(* IEC 61131-3 sources: AXOpen/src/components.festo.drives/ctrl/src/AxoCmmtAs (part 2) *)

                    IF Parametrization.Outputs.Done AND NOT Parametrization.Outputs.Error THEN
                        State := UINT#48;
                    END_IF;
                    IF Parametrization.Outputs.Error THEN
                        Messenger.Activate( UINT#1456, eAxoMessageCategory#Error);
                        MC_HomeErrorID :=   DINT#1456;
                        State := UINT#59;
                    END_IF;
                END_IF;
                IF State = UINT#48 THEN
                    Busy := TRUE;
                    Active := TRUE;
                    Parametrization.Inputs.Enable := FALSE;
                    IF  NOT Parametrization.Outputs.Done THEN
                        State := UINT#49;
                    END_IF;
                END_IF;
                //Write  PNU 11735 Homing mode
                IF State = UINT#49 THEN
                    Busy := TRUE;
                    Active := TRUE;
                    Parametrization.Inputs.Enable := TRUE;
                    Parametrization.Inputs.ReadWrite   := TRUE;
                    Parametrization.Inputs.ParameterNo := 11735;//mode
                    Parametrization.Inputs.Subindex    := 0;
                    Parametrization.Inputs.AxisNo  := BYTE#1;
                    Parametrization.Inputs.HardwareId  := _AxisReference^.HWIDs.HW_ModuleAccessPoint;
                    Parametrization.Inputs.ValueWriteLINT := TO_LINT(37);
                    IF Parametrization.Outputs.Done AND NOT Parametrization.Outputs.Error THEN
                        State := UINT#50;
                    END_IF;
                    IF Parametrization.Outputs.Error THEN
                        Messenger.Activate( UINT#1457, eAxoMessageCategory#Error);
                        MC_HomeErrorID :=   DINT#1457;
                        State := UINT#59;
                    END_IF;
                END_IF;
                IF State = UINT#50 THEN
                    Busy := TRUE;
                    Active := TRUE;
                    Parametrization.Inputs.Enable := FALSE;
                    IF  NOT Parametrization.Outputs.Done THEN
                        State := UINT#51;
                    END_IF;
                END_IF;
                //Homing started
                IF State = UINT#51 THEN
                    Busy := TRUE;
                    Active := TRUE;
                    _AxisReference^.Telegram111_Out.STW1.StartHoming := TRUE;
                    IF  NOT _AxisReference^.Telegram111_In.ZSW1.targetPosReached AND NOT _AxisReference^.Telegram111_In.ZSW1.homePosSet THEN
                        State := UINT#52;
                    END_IF;
                END_IF;
                IF State = UINT#52 THEN
                    Busy := TRUE;
                    Active := TRUE;
                    IF _AxisReference^.Telegram111_In.ZSW1.targetPosReached AND _AxisReference^.Telegram111_In.ZSW1.homePosSet THEN
                        _AxisReference^.Telegram111_Out.STW1.StartHoming := FALSE;
                        State := UINT#53;
                    END_IF;
                END_IF;
                //Write PNU 11203 Move to axis zero after homming
                IF State = UINT#53 THEN
                    Busy := TRUE;
                    Active := TRUE;
                    Parametrization.Inputs.Enable := TRUE;
                    Parametrization.Inputs.ReadWrite   := TRUE;
                    Parametrization.Inputs.ParameterNo := 11203;//Move to axis zero after homming
                    Parametrization.Inputs.Subindex    := 0;
                    Parametrization.Inputs.AxisNo  := BYTE#1;
                    Parametrization.Inputs.HardwareId  := _AxisReference^.HWIDs.HW_ModuleAccessPoint;
                    Parametrization.Inputs.ValueWriteBool := PNU_11203;
                    IF Parametrization.Outputs.Done AND NOT Parametrization.Outputs.Error THEN
                        State := UINT#54;
                    END_IF;
                    IF Parametrization.Outputs.Error THEN
                        Messenger.Activate( UINT#1458, eAxoMessageCategory#Error);
                        MC_HomeErrorID :=   DINT#1458;
                        State := UINT#59;
                    END_IF;
                END_IF;
                IF State = UINT#54 THEN
                    Busy := TRUE;
                    Active := TRUE;
                    Parametrization.Inputs.Enable := FALSE;
                    IF  NOT Parametrization.Outputs.Done THEN
                        State := UINT#55;
                    END_IF;
                END_IF;
                //Write PNU 11734 Axis zero point offset
                IF State = UINT#55 THEN
                    Busy := TRUE;
                    Active := TRUE;
                    Parametrization.Inputs.Enable := TRUE;
                    Parametrization.Inputs.ReadWrite   := TRUE;
                    Parametrization.Inputs.ParameterNo := 11734;//Move to axis zero after homming
                    Parametrization.Inputs.Subindex    := 0;
                    Parametrization.Inputs.AxisNo  := BYTE#1;
                    Parametrization.Inputs.HardwareId  := _AxisReference^.HWIDs.HW_ModuleAccessPoint;
                    Parametrization.Inputs.ValueWriteLINT := PNU_11734;
                    IF Parametrization.Outputs.Done AND NOT Parametrization.Outputs.Error THEN
                         State := UINT#56;
                    END_IF;
                    IF Parametrization.Outputs.Error THEN
                        Messenger.Activate( UINT#1459, eAxoMessageCategory#Error);
                        MC_HomeErrorID :=   DINT#1459;
                        State := UINT#59;
                    END_IF;
                END_IF;
                IF State = UINT#56 THEN
                    Busy := TRUE;
                    Active := TRUE;
                    Parametrization.Inputs.Enable := FALSE;
                    IF  NOT Parametrization.Outputs.Done THEN
                        State := UINT#57;
                    END_IF;
                END_IF;

                IF State = UINT#57 THEN
                    Parametrization.Inputs.Enable := TRUE;
                    Parametrization.Inputs.ReadWrite   := TRUE;
                    Parametrization.Inputs.ParameterNo := 11735;
                    Parametrization.Inputs.Subindex    := 0;
                    Parametrization.Inputs.AxisNo  := BYTE#1;
                    Parametrization.Inputs.HardwareId  := _AxisReference^.HWIDs.HW_ModuleAccessPoint;
                    Parametrization.Inputs.ValueWriteLINT := PNU_11735;

                    IF Parametrization.Outputs.Error THEN
                        Messenger.Activate( UINT#1460, eAxoMessageCategory#Error);
                        MC_HomeErrorID :=   DINT#1460;
                        State := UINT#59;
                    END_IF;
                    _AxisReference^.Telegram111_Out.STW1.StartHoming := FALSE;
                    Done := Parametrization.Outputs.Done AND NOT Parametrization.Outputs.Error;
                    MC_HomeCycle := ULINT#0;
                END_IF;
                IF State = UINT#58 THEN
                    _AxisReference^.Telegram111_Out.STW1.StartHoming := FALSE;
                    CommandAborted := TRUE;
                END_IF;
                IF State = UINT#59 THEN
                    _AxisReference^.Telegram111_Out.STW1.StartHoming := FALSE;
                    MC_HomeCycle := ULINT#0;
                    Error := TRUE;
                END_IF;

                IF State>=UINT#20 AND State<UINT#57 THEN
                    IF NOT _AxisReference^.Telegram111_In.ZSW1.operationEnabled THEN
                        State := UINT#58;
                    ELSIF _AxisReference^.Telegram111_In.ZSW1.faultPresent THEN
                        IF MC_HomeErrorID = DINT#0 THEN
                            MC_HomeErrorID := TO_DINT(_AxisReference^.Telegram111_In.Fault_Code);
                        END_IF;
                        State := UINT#59;
                    ELSIF _AxisReference^.Data.Cycle <> MC_HomeCycle THEN
                        _AxisReference^.Data.Cycle := _AxisReference^.Data.Cycle - ULINT#1;
                        State := UINT#58;
                    END_IF;
                END_IF;
                THIS.UpdateOutputs(AxisRef);
            END_IF;

            IF THIS.AxoHome_Task.DoneReached() THEN
                _AxisReference^.Status.CurrentMotionTaskId := AXOpen.Components.Drives.eAxoMotionTaskId#Axo_Done;
                MC_HomeErrorID := DINT#0;
                State := UINT#0;
                // MC_HomeCycle := ULINT#0;
                Parametrization.Inputs.Enable := FALSE;
                Parametrization.Inputs.ReadWrite   := FALSE;
                THIS.UpdateOutputs(AxisRef);
            END_IF;
            IF THIS.AxoHome_Task.RestoreTriggered() AND State>=UINT#20 AND State<=UINT#59 THEN
                _AxisReference^.Status.CurrentMotionTaskId := AXOpen.Components.Drives.eAxoMotionTaskId#Axo_None;
                MC_HomeErrorID := DINT#0;
                State := UINT#0;
                MC_HomeCycle := ULINT#0;
                Parametrization.Inputs.Enable := FALSE;
                Parametrization.Inputs.ReadWrite   := FALSE;
                THIS.UpdateOutputs(AxisRef);
            END_IF;

            ErrorID := MC_HomeErrorID;
            MC_HomeExecute_PV := Execute;
        END_METHOD

        ///<summary>
        /// This method commands a controlled motion stop and transfers the axis to the state ‘Stopping’. It aborts any
        /// ongoing method execution. While the axis is in state ‘Stopping’, no other method can perform any motion on the
        /// same axis.
        ///</summary>
        VAR INTERNAL
            MC_StopExecute_PV					: 	BOOL;				//Execute - previous value
            MC_StopErrorID					    : 	DINT;
            MC_StopCycle					    : 	ULINT;
        END_VAR
        METHOD PUBLIC OVERRIDE MC_Stop
            VAR_INPUT
                AxisRef         :   AXOpen.Components.Abstractions.Drives.IAxoAxisReference;
                Execute         :   BOOL;                       //  Start the action at rising edge
                Deceleration    :   LREAL;                      //  Value of the ‘Deceleration’ [u/s2]
                Jerk            :   LREAL;                      //  Value of the ‘Jerk’ [u/s3]
            END_VAR
            VAR_OUTPUT
                Done            :   BOOL;                       // Zero velocity reached
                Busy            :   BOOL;                       // The method is not finished and new output values are to be expected
                Active          :   BOOL;                       // Indicates that the method has control on the axis
                CommandAborted  :   BOOL;                       // ‘Command’ is aborted by switching off power (only possibility to abort)
                Error           :   BOOL;                       // Signals that an error has occurred within the method
                ErrorID         :   DINT;                       // Error identification
            END_VAR
            VAR
                _AxisReference :  REF_TO AXOpen.Components.Festo.Drives.AxoCmmtAsAxisReference;
            END_VAR

            _AxisReference ?= AxisRef;

            IF(_AxisReference = NULL) THEN
                Messenger.Activate(     UINT#1470, eAxoMessageCategory#ProgrammingError);
                DriveStatus.Error.Id := UINT#1470;
                RETURN;
            END_IF;

            Messenger.ActivateOnCondition(ULINT#1471, Execute AND Deceleration <= 0, eAxoMessageCategory#ProgrammingError);
            Messenger.ActivateOnCondition(ULINT#1472, Execute AND Jerk <= 0, eAxoMessageCategory#ProgrammingError);

            IF THIS.AxoStop_Task.StartTriggered() THEN
                _AxisReference^.Status.CurrentMotionTaskId := AXOpen.Components.Drives.eAxoMotionTaskId#Axo_Stop;
            END_IF;

            IF Execute AND NOT MC_StopExecute_PV THEN
                _AxisReference^.Data.Cycle := _AxisReference^.Data.Cycle + ULINT#2;
                MC_StopCycle := _AxisReference^.Data.Cycle ;
                State := UINT#0;
            END_IF;

            IF Execute THEN
                THIS.UpdateInputs(AxisRef);
                IF State = UINT#0 THEN
                    Busy := TRUE;
                    Active := TRUE;
                    MC_StopErrorID := DINT#0;
                    _AxisReference^.Telegram111_Out.STW2.TravelToFixStop := FALSE;
                    State := UINT#60;
                END_IF;

                IF State = UINT#60 THEN
                    IF Deceleration <= 0 OR Jerk <= 0 THEN
                        State := UINT#69;
                    ELSE
                        State := UINT#61;
                    END_IF;
                END_IF;
                //Writing PNU 12327 Jerk
                IF State = UINT#61 THEN
                    Busy := TRUE;
                    Active := TRUE;
                    Parametrization.Inputs.Enable := TRUE;
                    Parametrization.Inputs.ReadWrite   := TRUE;
                    Parametrization.Inputs.ParameterNo := 12327;
                    Parametrization.Inputs.Subindex    := 0;
                    Parametrization.Inputs.AxisNo  := BYTE#1;
                    Parametrization.Inputs.HardwareId  := _AxisReference^.HWIDs.HW_ModuleAccessPoint;
                    Parametrization.Inputs.ValueWriteREAL := TO_REAL(Jerk * ScalingConstantRequiredJerk );
                    IF Parametrization.Outputs.Done AND NOT Parametrization.Outputs.Error THEN
                        State := UINT#62;
                    END_IF;
                    IF Parametrization.Outputs.Error THEN
                        Messenger.Activate( UINT#1473, eAxoMessageCategory#Error);
                        MC_StopErrorID :=   DINT#1473;
                        State := UINT#69;
                    END_IF;
                END_IF;
                IF State = UINT#62 THEN
                    Busy := TRUE;
                    Active := TRUE;
                    _AxisReference^.Telegram111_Out.MDI_DEC := TO_UINT(Deceleration * ScalingConstantRequiredDeceleration);
                    _AxisReference^.Telegram111_Out.STW1.cancelTraversing := FALSE;
                    Parametrization.Inputs.Enable := FALSE;
                    Parametrization.Inputs.ReadWrite   := FALSE;
                    IF  NOT Parametrization.Outputs.Done THEN
                        State := UINT#63;
                    END_IF;
                END_IF;
                IF State = UINT#63 THEN
                    Busy := TRUE;
                    Active := TRUE;
                    IF _AxisReference^.Telegram111_In.ZSW1.driveStopped  THEN
                        State := UINT#64;
                    END_IF;
                END_IF;
                IF State = UINT#64 THEN
                    Busy := TRUE;
                    Active := TRUE;
                    IF TRUE THEN
                        State := UINT#65;
                    END_IF;
                END_IF;
                IF State = UINT#65 THEN
                    Busy := TRUE;
                    Active := TRUE;
                    IF TRUE THEN
                        State := UINT#66;
                    END_IF;
                END_IF;
                IF State = UINT#66 THEN
                    Busy := TRUE;
                    Active := TRUE;
                    IF TRUE THEN
                        State := UINT#67;
                    END_IF;
                END_IF;
                IF State = UINT#67 THEN
                    Done := TRUE;
                    Active := TRUE;
                    MC_StopCycle := ULINT#0;
                END_IF;
                IF State = UINT#68 THEN
                    CommandAborted := TRUE;
                END_IF;
                IF State = UINT#69 THEN
                    _AxisReference^.Telegram111_Out.MDI_DEC := UINT#16384;
                    _AxisReference^.Telegram111_Out.STW1.cancelTraversing := FALSE;
                    MC_StopCycle := ULINT#0;
                    Error := TRUE;
                END_IF;

                IF State>=UINT#60 AND State<UINT#67 THEN
                    IF NOT _AxisReference^.Telegram111_In.ZSW1.operationEnabled THEN
                        State := UINT#68;
                    ELSIF _AxisReference^.Telegram111_In.ZSW1.faultPresent THEN
                        IF MC_StopErrorID = DINT#0 THEN
                            MC_StopErrorID := TO_DINT(_AxisReference^.Telegram111_In.Fault_Code);
                        END_IF;
                        State := UINT#69;
                    ELSIF _AxisReference^.Data.Cycle <> MC_StopCycle THEN
                        _AxisReference^.Data.Cycle := _AxisReference^.Data.Cycle - ULINT#1;
                        State := UINT#68;
                    END_IF;
                END_IF;
                THIS.UpdateOutputs(AxisRef);
            END_IF;

            IF THIS.AxoStop_Task.DoneReached() THEN
                _AxisReference^.Status.CurrentMotionTaskId := AXOpen.Components.Drives.eAxoMotionTaskId#Axo_Done;
                _AxisReference^.Telegram111_Out.STW1.cancelTraversing := TRUE;
                MC_StopErrorID := DINT#0;
                State := UINT#0;
                // MC_StopCycle := ULINT#0;
                THIS.UpdateOutputs(AxisRef);
            END_IF;

            IF THIS.AxoStop_Task.RestoreTriggered() AND State>=UINT#60 AND State<=UINT#69 THEN
                _AxisReference^.Status.CurrentMotionTaskId := AXOpen.Components.Drives.eAxoMotionTaskId#Axo_None;
                _AxisReference^.Telegram111_Out.STW1.cancelTraversing := TRUE;
                MC_StopErrorID := DINT#0;
                State := UINT#0;
                MC_StopCycle := ULINT#0;
                THIS.UpdateOutputs(AxisRef);
            END_IF;

            ErrorID := MC_StopErrorID;
            MC_StopExecute_PV := Execute;
        END_METHOD

        ///<summary>
        /// This method commands a controlled motion stop. The axis is moved to the state ‘DiscreteMotion’, until the
        /// velocity is zero. With the ‘Done’ output set, the state is transferred to ‘Standstill’.
        ///</summary>
        VAR INTERNAL
            MC_HaltExecute_PV					: 	BOOL;				//Execute - previous value
            MC_HaltErrorID					    : 	DINT;
            MC_HaltCycle					    : 	ULINT;
        END_VAR
        METHOD PUBLIC OVERRIDE MC_Halt
            VAR_INPUT
                AxisRef         :   AXOpen.Components.Abstractions.Drives.IAxoAxisReference;
                Execute         :   BOOL;                       //  Start the action at rising edge
                Deceleration    :   LREAL;                      //  Value of the ‘Deceleration’ [u/s2]
                Jerk            :   LREAL;                      //  Value of the ‘Jerk’ [u/s3]
            END_VAR
            VAR_OUTPUT
                Done            :   BOOL;                       // Zero velocity reached
                Busy            :   BOOL;                       // The method is not finished and new output values are to be expected
                Active          :   BOOL;                       // Indicates that the method has control on the axis
                CommandAborted  :   BOOL;                       // ‘Command’ is aborted by switching off power (only possibility to abort)
                Error           :   BOOL;                       // Signals that an error has occurred within the method
                ErrorID         :   DINT;                       // Error identification
            END_VAR
            VAR
                _AxisReference :  REF_TO AXOpen.Components.Festo.Drives.AxoCmmtAsAxisReference;
            END_VAR

            _AxisReference ?= AxisRef;

            IF(_AxisReference = NULL) THEN
                Messenger.Activate(     UINT#1480, eAxoMessageCategory#ProgrammingError);
                DriveStatus.Error.Id := UINT#1480;
                RETURN;
            END_IF;

            IF THIS.AxoHalt_Task.StartTriggered() THEN
                _AxisReference^.Status.CurrentMotionTaskId := AXOpen.Components.Drives.eAxoMotionTaskId#Axo_Halt;
            END_IF;

            IF Execute AND NOT MC_HaltExecute_PV THEN
                _AxisReference^.Data.Cycle := _AxisReference^.Data.Cycle + ULINT#2;
                MC_HaltCycle := _AxisReference^.Data.Cycle ;
                State := UINT#0;
            END_IF;

            IF Execute THEN
                Messenger.ActivateOnCondition(ULINT#1481, Execute AND Deceleration <= 0, eAxoMessageCategory#ProgrammingError);
                Messenger.ActivateOnCondition(ULINT#1482, Execute AND Jerk <= 0, eAxoMessageCategory#ProgrammingError);

                THIS.UpdateInputs(AxisRef);
                IF State = UINT#0 THEN
                    Busy := TRUE;
                    Active := TRUE;
                    MC_HaltErrorID := DINT#0;
                    _AxisReference^.Telegram111_Out.STW2.TravelToFixStop := FALSE;
                    State := UINT#70;
                END_IF;

                IF State = UINT#70 THEN
                    IF Deceleration <= 0 OR Jerk <= 0 THEN
                        State := UINT#79;
                    ELSE
                        State := UINT#71;
                    END_IF;
                END_IF;
                IF State = UINT#71 THEN
                    Busy := TRUE;
                    Active := TRUE;
                    Parametrization.Inputs.Enable := TRUE;
                    Parametrization.Inputs.ReadWrite   := TRUE;
                    Parametrization.Inputs.ParameterNo := 12327;
                    Parametrization.Inputs.Subindex    := 0;
                    Parametrization.Inputs.AxisNo  := BYTE#1;
                    Parametrization.Inputs.HardwareId  := _AxisReference^.HWIDs.HW_ModuleAccessPoint;
                    Parametrization.Inputs.ValueWriteREAL := TO_REAL(Jerk * ScalingConstantRequiredJerk);
                    IF Parametrization.Outputs.Done AND NOT Parametrization.Outputs.Error THEN
                        State := UINT#72;
                    END_IF;
                    IF Parametrization.Outputs.Error THEN
                        Messenger.Activate( UINT#1483, eAxoMessageCategory#Error);
                        MC_HaltErrorID :=   DINT#1483;
                        State := UINT#79;
                    END_IF;
                END_IF;
                IF State = UINT#72 THEN
                    Busy := TRUE;
                    Active := TRUE;
                    _AxisReference^.Telegram111_Out.MDI_DEC := TO_UINT(Deceleration * ScalingConstantRequiredDeceleration);
                    _AxisReference^.Telegram111_Out.STW1.cancelTraversing := FALSE;
                    Parametrization.Inputs.Enable := FALSE;
                    Parametrization.Inputs.ReadWrite   := FALSE;
                    IF  NOT Parametrization.Outputs.Done THEN
                        State := UINT#73;
                    END_IF;
                END_IF;
                IF State = UINT#73 THEN
                    Busy := TRUE;
                    Active := TRUE;
                    IF _AxisReference^.Telegram111_In.ZSW1.driveStopped  THEN
                        State := UINT#74;
                    END_IF;
                END_IF;
                IF State = UINT#74 THEN
                    IF TRUE THEN
                        State := UINT#75;
                    END_IF;
                END_IF;
                IF State = UINT#75 THEN
                    IF TRUE THEN
                        State := UINT#76;
                    END_IF;
                END_IF;
                IF State = UINT#76 THEN
                    IF TRUE THEN
                        State := UINT#77;
                    END_IF;
                END_IF;
                IF State = UINT#77 THEN
                    Done := TRUE;
                    _AxisReference^.Telegram111_Out.STW1.cancelTraversing := TRUE;
                    MC_HaltCycle := ULINT#0;
                END_IF;
                IF State = UINT#78 THEN
                    _AxisReference^.Telegram111_Out.STW1.cancelTraversing := TRUE;
                    CommandAborted := TRUE;
                END_IF;
                IF State = UINT#79 THEN
                    _AxisReference^.Telegram111_Out.MDI_DEC := UINT#16384;
                    _AxisReference^.Telegram111_Out.STW1.cancelTraversing := FALSE;
                    MC_HaltCycle := ULINT#0;
                    Error := TRUE;
                END_IF;

                IF State>=UINT#70 AND State<UINT#77 THEN
                    IF NOT _AxisReference^.Telegram111_In.ZSW1.operationEnabled THEN
                        State := UINT#78;
                    ELSIF _AxisReference^.Telegram111_In.ZSW1.faultPresent THEN
                        IF MC_HaltErrorID = DINT#0 THEN
                            MC_HaltErrorID := TO_DINT(_AxisReference^.Telegram111_In.Fault_Code);
                        END_IF;
                        State := UINT#79;
                    ELSIF _AxisReference^.Data.Cycle <> MC_HaltCycle THEN
                        _AxisReference^.Data.Cycle := _AxisReference^.Data.Cycle - ULINT#1;
                        State := UINT#78;
                    END_IF;
                END_IF;
                THIS.UpdateOutputs(AxisRef);
            END_IF;

            IF THIS.AxoHalt_Task.DoneReached() THEN
                _AxisReference^.Status.CurrentMotionTaskId := AXOpen.Components.Drives.eAxoMotionTaskId#Axo_Done;
                _AxisReference^.Telegram111_Out.STW1.cancelTraversing := TRUE;
                MC_HaltErrorID := DINT#0;
                State := UINT#0;
                // MC_HaltCycle := ULINT#0;
                THIS.UpdateOutputs(AxisRef);
            END_IF;

            IF THIS.AxoHalt_Task.RestoreTriggered() AND State>=UINT#70 AND State<=UINT#79 THEN
                _AxisReference^.Status.CurrentMotionTaskId := AXOpen.Components.Drives.eAxoMotionTaskId#Axo_None;
                _AxisReference^.Telegram111_Out.STW1.cancelTraversing := TRUE;
                MC_HaltErrorID := DINT#0;
                State := UINT#0;
                MC_HaltCycle := ULINT#0;
                THIS.UpdateOutputs(AxisRef);
            END_IF;

            ErrorID := MC_HaltErrorID;
            MC_HaltExecute_PV := Execute;
        END_METHOD

        ///<summary>
        /// This method commands a controlled motion to a specified absolute position.
        ///</summary>
        VAR INTERNAL
            MC_MoveAbsoluteExecute_PV					: 	BOOL;				//Execute - previous value
            MC_MoveAbsoluteErrorID					    : 	DINT;
            MC_MoveAbsoluteCycle					    : 	ULINT;
            MC_MoveAbsoluteContinuousUpdate_SV          :   BOOL;
            MC_MoveAbsolutePosition_PV                  :   LREAL;
            MC_MoveAbsoluteVelocity_PV                  :   LREAL;
            MC_MoveAbsoluteAcceleration_PV              :   LREAL;
            MC_MoveAbsoluteDeceleration_PV              :   LREAL;
            MC_MoveAbsoluteJerk_PV                      :   LREAL;
            MC_MoveAbsoluteDirection_PV                 :   AXOpen.Components.Abstractions.Drives.eAxoDriveDirection;
        END_VAR
        METHOD PUBLIC OVERRIDE MC_MoveAbsolute
            VAR_INPUT
                AxisRef         :   AXOpen.Components.Abstractions.Drives.IAxoAxisReference;
                Execute         :   BOOL;                       //  Start the motion at rising edge
                ContinuousUpdate:   BOOL;                       //  Activate ‘ContinuousUpdate’ - target parameters should be changed during movement
                Position        :   LREAL;                      //  Commanded ‘Position’ for the motion (in technical unit [u]) (negative or positive)
                Velocity        :   LREAL;                      //  Value of the maximum ‘Velocity’ (not necessarily reached) [u/s].
                Acceleration    :   LREAL;                      //  Value of the ‘Acceleration’ (always positive) (increasing energy of the motor) [u/s2]
                Deceleration    :   LREAL;                      //  Value of the ‘Deceleration’ (always positive) (decreasing energy of the motor) [u/s2]
                Jerk            :   LREAL;                      //  Value of the ‘Jerk’ [u/s3]
                Direction       :   AXOpen.Components.Abstractions.Drives.eAxoDriveDirection;         //  Enum type (1-of-4 values: PositiveDirection, ShortestWay, NegativeDirection, CurrentDirection)
            END_VAR
            VAR_OUTPUT
                Done            :   BOOL;                       // Commanded position finally reached
                Busy            :   BOOL;                       // The method is not finished and new output values are to be expected
                Active          :   BOOL;                       // Indicates that the method has control on the axis
                CommandAborted  :   BOOL;                       // ‘Command’ is aborted by another command
                Error           :   BOOL;                       // Signals that an error has occurred within the method
                ErrorID         :   DINT;                       // Error identification
            END_VAR
            VAR
                _AxisReference :  REF_TO AXOpen.Components.Festo.Drives.AxoCmmtAsAxisReference;
                Dummy : BOOL;
            END_VAR

            _AxisReference ?= AxisRef;

            IF(_AxisReference = NULL) THEN
                Messenger.Activate(     UINT#1490, eAxoMessageCategory#ProgrammingError);
                DriveStatus.Error.Id := UINT#1490;
                RETURN;
            END_IF;

            Messenger.ActivateOnCondition(ULINT#1491, Execute AND Velocity <= 0, eAxoMessageCategory#ProgrammingError);
            Messenger.ActivateOnCondition(ULINT#1492, Execute AND Acceleration <= 0, eAxoMessageCategory#ProgrammingError);
            Messenger.ActivateOnCondition(ULINT#1493, Execute AND Deceleration <= 0, eAxoMessageCategory#ProgrammingError);
            Messenger.ActivateOnCondition(ULINT#1494, Execute AND Jerk <= 0, eAxoMessageCategory#ProgrammingError);

            IF THIS.AxoMoveAbsolute_Task.StartTriggered()  THEN
                _AxisReference^.Status.CurrentMotionTaskId := AXOpen.Components.Drives.eAxoMotionTaskId#Axo_MoveAbsolute;
            END_IF;

            IF Execute AND NOT MC_MoveAbsoluteExecute_PV AND State = UINT#0 THEN
                _AxisReference^.Data.Cycle := _AxisReference^.Data.Cycle + ULINT#2;
                MC_MoveAbsoluteCycle := _AxisReference^.Data.Cycle ;
            END_IF;

            IF Execute THEN
                THIS.UpdateInputs(AxisRef);

                IF NOT ContinuousUpdate THEN
                    MC_MoveAbsoluteContinuousUpdate_SV := FALSE;
                END_IF;

                IF State = UINT#0 THEN
                    Busy := TRUE;
                    Active := TRUE;
                    MC_MoveAbsoluteErrorID := DINT#0;
                    _AxisReference^.Telegram111_Out.STW1.StartHoming := FALSE;
                    _AxisReference^.Telegram111_Out.POS_STW1.MDI_MOD := FALSE;
                    _AxisReference^.Telegram111_Out.POS_STW1.PosModulo := FALSE;
                    _AxisReference^.Telegram111_Out.POS_STW1.NegModulo := FALSE;
                    _AxisReference^.Telegram111_Out.POS_STW1.SetupMode := FALSE;
                    _AxisReference^.Telegram111_Out.POS_STW1.MDI_Activate := FALSE;
                    _AxisReference^.Telegram111_Out.POS_STW2.Trackingmode := FALSE;
                    _AxisReference^.Telegram111_Out.POS_STW2.jog_inc := FALSE;
                    _AxisReference^.Telegram111_Out.POS_STW1.travBlockBit0 := FALSE;
                    _AxisReference^.Telegram111_Out.POS_STW1.travBlockBit1 := FALSE;
                    _AxisReference^.Telegram111_Out.POS_STW1.travBlockBit2 := FALSE;
                    _AxisReference^.Telegram111_Out.POS_STW1.travBlockBit3 := FALSE;
                    _AxisReference^.Telegram111_Out.POS_STW1.travBlockBit4 := FALSE;
                    _AxisReference^.Telegram111_Out.POS_STW1.travBlockBit5 := FALSE;
                    _AxisReference^.Telegram111_Out.POS_STW1.travBlockBit6 := FALSE;
                    _AxisReference^.Telegram111_Out.STW2.TravelToFixStop := FALSE;
                    Parametrization.Inputs.Enable := FALSE;
                    MC_MoveAbsoluteContinuousUpdate_SV := ContinuousUpdate;
                    State := UINT#80;
                END_IF;
                IF State = UINT#80 THEN
                    Busy := TRUE;
                    Active := TRUE;
                    IF Velocity > 0 AND Acceleration > 0 AND Deceleration >0 AND Jerk > 0 THEN
                        _AxisReference^.Telegram111_Out.MDI_TARPOS :=       TO_DINT(Position        *   ScalingConstantRequiredPosition);
                        _AxisReference^.Telegram111_Out.MDI_VELOCITY :=     TO_DINT(Velocity        *   ScalingConstantRequiredVelocity     * _AxisReference^.Data.OverrideVelocityFactor);
                        _AxisReference^.Telegram111_Out.MDI_ACC :=          TO_UINT(Acceleration    *   ScalingConstantRequiredAcceleration * _AxisReference^.Data.OverrideAccelerationFactor);
                        _AxisReference^.Telegram111_Out.MDI_DEC :=          TO_UINT(Deceleration    *   ScalingConstantRequiredDeceleration * _AxisReference^.Data.OverrideAccelerationFactor);
                        MC_MoveAbsolutePosition_PV      :=  Position;
                        MC_MoveAbsoluteVelocity_PV      :=  Velocity;
                        MC_MoveAbsoluteAcceleration_PV  :=  Acceleration;
                        MC_MoveAbsoluteDeceleration_PV  :=  Deceleration;
                        MC_MoveAbsoluteJerk_PV          :=  Jerk;
                        MC_MoveAbsoluteDirection_PV     :=  Direction;
                        State := UINT#81;
                    END_IF;
                END_IF;
                //Writing PNU 12327 Jerk
                IF State = UINT#81 THEN
                    Busy := TRUE;
                    Active := TRUE;
                    Parametrization.Inputs.Enable := TRUE;
                    Parametrization.Inputs.ReadWrite   := TRUE;
                    Parametrization.Inputs.ParameterNo := 12327;
                    Parametrization.Inputs.Subindex    := 0;
                    Parametrization.Inputs.AxisNo  := BYTE#1;
                    Parametrization.Inputs.HardwareId  := _AxisReference^.HWIDs.HW_ModuleAccessPoint;
                    Parametrization.Inputs.ValueWriteREAL := TO_REAL(MC_MoveAbsoluteJerk_PV * ScalingConstantRequiredJerk * _AxisReference^.Data.OverrideJerkFactor);
                    IF Parametrization.Outputs.Done AND NOT Parametrization.Outputs.Error THEN
                        State := UINT#82;
                    END_IF;
                    IF Parametrization.Outputs.Error THEN
                        Messenger.Activate(         UINT#1495, eAxoMessageCategory#Error);
                        MC_MoveAbsoluteErrorID :=   DINT#1495;
                        State := UINT#89;
                    END_IF;
                END_IF;
                IF State = UINT#82 THEN
                    Busy := TRUE;
                    Active := TRUE;
                    Parametrization.Inputs.Enable := FALSE;
                    Parametrization.Inputs.ReadWrite   := FALSE;
                    IF  NOT Parametrization.Outputs.Done THEN
                        State := UINT#83;
                    END_IF;
                END_IF;
                //Executing movement
                IF State = UINT#83 THEN
                    _AxisReference^.Telegram111_Out.POS_STW1.MDI_Activate := TRUE;
                    _AxisReference^.Telegram111_Out.POS_STW1.MDI_MOD := TRUE;
                    _AxisReference^.Telegram111_Out.STW1.activateTraversing := TRUE;
                    IF _AxisReference^.Telegram111_In.ZSW1.acknowledgeTraversingBlockActivated THEN
                        State := UINT#84;
                    END_IF;
                END_IF;
                IF State = UINT#84 THEN
                    _AxisReference^.Telegram111_Out.STW1.activateTraversing := FALSE;
                    IF _AxisReference^.Telegram111_In.ZSW1.targetPosReached
                        AND ABS( Position - THIS.ActualPosition) <=  _AxisReference^.Config.InPositionWindow THEN
                        State := UINT#85;
                    END_IF;
                END_IF;
                IF State = UINT#85 THEN
                    IF TRUE THEN
                        State := UINT#86;
                    END_IF;
                END_IF;
                IF State = UINT#86 THEN
                    IF TRUE THEN
                        State := UINT#87;
                    END_IF;
                END_IF;
                IF State = UINT#87 THEN
                    Done := TRUE;
                    MC_MoveAbsoluteCycle := ULINT#0;
                END_IF;
                IF State = UINT#88 THEN
                    CommandAborted := TRUE;
                END_IF;
                IF State = UINT#89 THEN
                    MC_MoveAbsoluteCycle := ULINT#0;
                    Error := TRUE;
                END_IF;

                IF State>=UINT#80 AND State<UINT#87 THEN
                    IF MC_MoveAbsoluteContinuousUpdate_SV AND (
                        MC_MoveAbsolutePosition_PV      <>  Position OR
                        MC_MoveAbsoluteVelocity_PV      <>  Velocity OR
                        MC_MoveAbsoluteAcceleration_PV  <>  Acceleration OR
                        MC_MoveAbsoluteDeceleration_PV  <>  Deceleration OR
                        MC_MoveAbsoluteJerk_PV          <>  Jerk OR
                        MC_MoveAbsoluteDirection_PV     <>  Direction ) THEN
                        _AxisReference^.Telegram111_Out.STW1.activateTraversing := FALSE;
                        IF NOT _AxisReference^.Telegram111_In.ZSW1.acknowledgeTraversingBlockActivated THEN
                            State := UINT#80;
                        END_IF;
                    END_IF;
                    IF NOT _AxisReference^.Telegram111_In.ZSW1.operationEnabled THEN
                        State := UINT#88;
                    ELSIF _AxisReference^.Telegram111_In.ZSW1.faultPresent THEN
                        IF MC_MoveAbsoluteErrorID = DINT#0 THEN
                            MC_MoveAbsoluteErrorID := TO_DINT(_AxisReference^.Telegram111_In.Fault_Code);
                        END_IF;
                        State := UINT#89;
                    ELSIF _AxisReference^.Data.Cycle <> MC_MoveAbsoluteCycle THEN
                        _AxisReference^.Data.Cycle := _AxisReference^.Data.Cycle - ULINT#1;
                        State := UINT#88;
                    END_IF;
                END_IF;

                THIS.UpdateOutputs(AxisRef);
            END_IF;

            IF THIS.AxoMoveAbsolute_Task.DoneReached() THEN
                _AxisReference^.Status.CurrentMotionTaskId := AXOpen.Components.Drives.eAxoMotionTaskId#Axo_Done;
                _AxisReference^.Telegram111_Out.STW1.activateTraversing := FALSE;
                MC_MoveAbsoluteErrorID := DINT#0;
                State := UINT#0;
                // MC_MoveAbsoluteCycle := ULINT#0;
                THIS.UpdateOutputs(AxisRef);
            END_IF;

            IF THIS.AxoMoveAbsolute_Task.RestoreTriggered() AND State>=UINT#80 AND State<=UINT#89 THEN
                _AxisReference^.Status.CurrentMotionTaskId := AXOpen.Components.Drives.eAxoMotionTaskId#Axo_None;
                _AxisReference^.Telegram111_Out.STW1.activateTraversing := FALSE;
                MC_MoveAbsoluteErrorID := DINT#0;
                MC_MoveAbsoluteCycle := ULINT#0;
                State := UINT#0;
                MC_MoveAbsoluteExecute_PV := FALSE;
                THIS.UpdateOutputs(AxisRef);
            END_IF;

            ErrorID := MC_MoveAbsoluteErrorID;
            MC_MoveAbsoluteExecute_PV := Execute;
        END_METHOD

        ///<summary>
        /// This method  commands a controlled motion of a specified distance relative to the set position at the time of the execution.
        ///</summary>
        VAR INTERNAL
            MC_MoveRelativeExecute_PV					: 	BOOL;				//Execute - previous value
            MC_MoveRelativeErrorID					    : 	DINT;
            MC_MoveRelativeCycle					    : 	ULINT;
            MC_MoveRelativeContinuousUpdate_SV          :   BOOL;
            MC_MoveRelativeDistance_PV                  :   LREAL;
            MC_MoveRelativeVelocity_PV                  :   LREAL;
            MC_MoveRelativeAcceleration_PV              :   LREAL;
            MC_MoveRelativeDeceleration_PV              :   LREAL;
            MC_MoveRelativeJerk_PV                      :   LREAL;
        END_VAR
        METHOD PUBLIC OVERRIDE MC_MoveRelative
            VAR_INPUT
                AxisRef         :   AXOpen.Components.Abstractions.Drives.IAxoAxisReference;
                Execute         :   BOOL;                       //  Start the motion at rising edge
                ContinuousUpdate:   BOOL;                       //  Activate ‘ContinuousUpdate’ - target parameters should be changed during movement
                Distance        :   LREAL;                      //  Relative distance for the motion (in technical unit [u]
                Velocity        :   LREAL;                      //  Value of the maximum ‘Velocity’ (not necessarily reached) [u/s].
                Acceleration    :   LREAL;                      //  Value of the ‘Acceleration’ (always positive) (increasing energy of the motor) [u/s2]
                Deceleration    :   LREAL;                      //  Value of the ‘Deceleration’ (always positive) (decreasing energy of the motor) [u/s2]
                Jerk            :   LREAL;                      //  Value of the ‘Jerk’ [u/s3]
            END_VAR
            VAR_OUTPUT
                Done            :   BOOL;                       // Commanded distance reached
                Busy            :   BOOL;                       // The method is not finished and new output values are to be expected
                Active          :   BOOL;                       // Indicates that the method has control on the axis
                CommandAborted  :   BOOL;                       // ‘Command’ is aborted by another command
                Error           :   BOOL;                       // Signals that an error has occurred within the method
                ErrorID         :   DINT;                       // Error identification
            END_VAR
            VAR
                _AxisReference :  REF_TO AXOpen.Components.Festo.Drives.AxoCmmtAsAxisReference;
                Dummy : BOOL;
            END_VAR

            _AxisReference ?= AxisRef;

            IF(_AxisReference = NULL) THEN
                Messenger.Activate(     UINT#1500, eAxoMessageCategory#ProgrammingError);
                DriveStatus.Error.Id := UINT#1500;
                RETURN;
            END_IF;

            Messenger.ActivateOnCondition(ULINT#1501, Execute AND Velocity <= 0, eAxoMessageCategory#ProgrammingError);
            Messenger.ActivateOnCondition(ULINT#1502, Execute AND Acceleration <= 0, eAxoMessageCategory#ProgrammingError);
            Messenger.ActivateOnCondition(ULINT#1503, Execute AND Deceleration <= 0, eAxoMessageCategory#ProgrammingError);
            Messenger.ActivateOnCondition(ULINT#1504, Execute AND Jerk <= 0, eAxoMessageCategory#ProgrammingError);

            IF THIS.AxoMoveRelative_Task.StartTriggered()  THEN
                _AxisReference^.Status.CurrentMotionTaskId := AXOpen.Components.Drives.eAxoMotionTaskId#Axo_MoveRelative;
            END_IF;

            IF Execute AND NOT MC_MoveRelativeExecute_PV AND State = UINT#0 THEN
                _AxisReference^.Data.Cycle := _AxisReference^.Data.Cycle + ULINT#2;
                MC_MoveRelativeCycle := _AxisReference^.Data.Cycle ;
            END_IF;

            IF Execute THEN
                THIS.UpdateInputs(AxisRef);
                IF NOT ContinuousUpdate THEN
                    MC_MoveRelativeContinuousUpdate_SV := FALSE;
                END_IF;

                IF State = UINT#0 THEN
                    Busy := TRUE;
                    Active := TRUE;
                    MC_MoveRelativeErrorID := DINT#0;
                    _AxisReference^.Telegram111_Out.STW1.StartHoming := FALSE;
                    _AxisReference^.Telegram111_Out.POS_STW1.MDI_MOD := FALSE;
                    _AxisReference^.Telegram111_Out.POS_STW1.PosModulo := FALSE;
                    _AxisReference^.Telegram111_Out.POS_STW1.NegModulo := FALSE;
                    _AxisReference^.Telegram111_Out.POS_STW1.SetupMode := FALSE;
                    _AxisReference^.Telegram111_Out.POS_STW1.MDI_Activate := FALSE;
                    _AxisReference^.Telegram111_Out.POS_STW2.Trackingmode := FALSE;
                    _AxisReference^.Telegram111_Out.POS_STW2.jog_inc := FALSE;
                    _AxisReference^.Telegram111_Out.POS_STW1.travBlockBit0 := FALSE;
                    _AxisReference^.Telegram111_Out.POS_STW1.travBlockBit1 := FALSE;
                    _AxisReference^.Telegram111_Out.POS_STW1.travBlockBit2 := FALSE;
                    _AxisReference^.Telegram111_Out.POS_STW1.travBlockBit3 := FALSE;
                    _AxisReference^.Telegram111_Out.POS_STW1.travBlockBit4 := FALSE;
                    _AxisReference^.Telegram111_Out.POS_STW1.travBlockBit5 := FALSE;
                    _AxisReference^.Telegram111_Out.POS_STW1.travBlockBit6 := FALSE;
                    _AxisReference^.Telegram111_Out.STW2.TravelToFixStop := FALSE;
                    Parametrization.Inputs.Enable := FALSE;
                    MC_MoveRelativeContinuousUpdate_SV := ContinuousUpdate;
                    State := UINT#90;
                END_IF;
                IF State = UINT#90 THEN
                    Busy := TRUE;
                    Active := TRUE;
                    IF Velocity > 0 AND Acceleration > 0 AND Deceleration >0 AND Jerk > 0 THEN
                        _AxisReference^.Telegram111_Out.MDI_TARPOS :=       TO_DINT(Distance        *   ScalingConstantRequiredPosition);
                        _AxisReference^.Telegram111_Out.MDI_VELOCITY :=     TO_DINT(Velocity        *   ScalingConstantRequiredVelocity     * _AxisReference^.Data.OverrideVelocityFactor);
                        _AxisReference^.Telegram111_Out.MDI_ACC :=          TO_UINT(Acceleration    *   ScalingConstantRequiredAcceleration * _AxisReference^.Data.OverrideAccelerationFactor);
                        _AxisReference^.Telegram111_Out.MDI_DEC :=          TO_UINT(Deceleration    *   ScalingConstantRequiredDeceleration * _AxisReference^.Data.OverrideAccelerationFactor);
                        MC_MoveRelativeDistance_PV      :=  Distance;
                        MC_MoveRelativeVelocity_PV      :=  Velocity;
                        MC_MoveRelativeAcceleration_PV  :=  Acceleration;
                        MC_MoveRelativeDeceleration_PV  :=  Deceleration;
                        MC_MoveRelativeJerk_PV          :=  Jerk;
                        State := UINT#91;
                    END_IF;
                END_IF;
                //Writing PNU 12327 Jerk
                IF State = UINT#91 THEN
                    Busy := TRUE;
                    Active := TRUE;
                    Parametrization.Inputs.Enable := TRUE;
                    Parametrization.Inputs.ReadWrite   := TRUE;
                    Parametrization.Inputs.ParameterNo := 12327;
                    Parametrization.Inputs.Subindex    := 0;
                    Parametrization.Inputs.AxisNo  := BYTE#1;
                    Parametrization.Inputs.HardwareId  := _AxisReference^.HWIDs.HW_ModuleAccessPoint;
                    Parametrization.Inputs.ValueWriteREAL := TO_REAL(MC_MoveRelativeJerk_PV  * ScalingConstantRequiredJerk * _AxisReference^.Data.OverrideJerkFactor);
                    IF Parametrization.Outputs.Done AND NOT Parametrization.Outputs.Error THEN
                        State := UINT#92;
                    END_IF;
                    IF Parametrization.Outputs.Error THEN
                        Messenger.Activate(         UINT#1505, eAxoMessageCategory#Error);
                        MC_MoveRelativeErrorID :=   DINT#1505;
                        State := UINT#99;
                    END_IF;
                END_IF;
                IF State = UINT#92 THEN
                    Busy := TRUE;
                    Active := TRUE;
                    Parametrization.Inputs.Enable := FALSE;
                    Parametrization.Inputs.ReadWrite   := FALSE;
                    IF  NOT Parametrization.Outputs.Done THEN
                        State := UINT#93;
                    END_IF;
                END_IF;
                //Executing movement
                IF State = UINT#93 THEN
                    _AxisReference^.Telegram111_Out.POS_STW1.MDI_Activate := TRUE;
                    _AxisReference^.Telegram111_Out.POS_STW1.MDI_MOD := FALSE;
                    _AxisReference^.Telegram111_Out.STW1.activateTraversing := TRUE;
                    IF _AxisReference^.Telegram111_In.ZSW1.acknowledgeTraversingBlockActivated THEN
                        State := UINT#94;
                    END_IF;
                END_IF;
                IF State = UINT#94 THEN
                    _AxisReference^.Telegram111_Out.STW1.activateTraversing := FALSE;
                    IF _AxisReference^.Telegram111_In.ZSW1.targetPosReached THEN
                        State := UINT#95;
                    END_IF;
                END_IF;
                IF State = UINT#95 THEN
                    IF TRUE THEN
                        State := UINT#96;
                    END_IF;
                END_IF;
                IF State = UINT#96 THEN
                    IF TRUE THEN
                        State := UINT#97;
                    END_IF;
                END_IF;
                IF State = UINT#97 THEN
                    Done := TRUE;
                    MC_MoveRelativeCycle := ULINT#0;
                END_IF;
                IF State = UINT#98 THEN
                    CommandAborted := TRUE;
                END_IF;
                IF State = UINT#99 THEN
                    MC_MoveRelativeCycle := ULINT#0;
                    Error := TRUE;
                END_IF;

                IF State>=UINT#90 AND State<UINT#97 THEN
                    IF MC_MoveRelativeContinuousUpdate_SV AND (
                        MC_MoveRelativeDistance_PV      <>  Distance OR
                        MC_MoveRelativeVelocity_PV      <>  Velocity OR
                        MC_MoveRelativeAcceleration_PV  <>  Acceleration OR
                        MC_MoveRelativeDeceleration_PV  <>  Deceleration OR
                        MC_MoveRelativeJerk_PV          <>  Jerk ) THEN
                        _AxisReference^.Telegram111_Out.STW1.activateTraversing := FALSE;
                        IF NOT _AxisReference^.Telegram111_In.ZSW1.acknowledgeTraversingBlockActivated THEN
                            _AxisReference^.Telegram111_Out.MDI_TARPOS :=   TO_DINT((Distance)      *   ScalingConstantRequiredPosition) - _AxisReference^.Telegram111_In.XIST_A;
                            _AxisReference^.Telegram111_Out.MDI_VELOCITY := TO_DINT(Velocity        *   ScalingConstantRequiredVelocity     * _AxisReference^.Data.OverrideVelocityFactor);
                            _AxisReference^.Telegram111_Out.MDI_ACC :=      TO_UINT(Acceleration    *   ScalingConstantRequiredAcceleration * _AxisReference^.Data.OverrideAccelerationFactor);
                            _AxisReference^.Telegram111_Out.MDI_DEC :=      TO_UINT(Deceleration    *   ScalingConstantRequiredDeceleration * _AxisReference^.Data.OverrideAccelerationFactor);
                            MC_MoveRelativeDistance_PV      :=  Distance;
                            MC_MoveRelativeVelocity_PV      :=  Velocity;
                            MC_MoveRelativeAcceleration_PV  :=  Acceleration;
                            MC_MoveRelativeDeceleration_PV  :=  Deceleration;
                            MC_MoveRelativeJerk_PV          :=  Jerk;
                            State := UINT#91;
                        END_IF;
                    END_IF;
                    IF NOT _AxisReference^.Telegram111_In.ZSW1.operationEnabled THEN
                        State := UINT#98;
                    ELSIF _AxisReference^.Telegram111_In.ZSW1.faultPresent THEN
                        IF MC_MoveRelativeErrorID = DINT#0 THEN
                            MC_MoveRelativeErrorID := TO_DINT(_AxisReference^.Telegram111_In.Fault_Code);
                        END_IF;
                        State := UINT#99;
                    ELSIF _AxisReference^.Data.Cycle <> MC_MoveRelativeCycle THEN
                        _AxisReference^.Data.Cycle := _AxisReference^.Data.Cycle - ULINT#1;
                        State := UINT#98;
                    END_IF;
                END_IF;
                THIS.UpdateOutputs(AxisRef);
            END_IF;

            IF THIS.AxoMoveRelative_Task.DoneReached() THEN
                _AxisReference^.Status.CurrentMotionTaskId := AXOpen.Components.Drives.eAxoMotionTaskId#Axo_Done;
                _AxisReference^.Telegram111_Out.STW1.activateTraversing := FALSE;
                MC_MoveRelativeErrorID := DINT#0;
                // MC_MoveRelativeCycle := ULINT#0;
                State := UINT#0;
                THIS.UpdateOutputs(AxisRef);
            END_IF;

            IF THIS.AxoMoveRelative_Task.RestoreTriggered() AND State>=UINT#90 AND State<=UINT#99 THEN
                _AxisReference^.Status.CurrentMotionTaskId := AXOpen.Components.Drives.eAxoMotionTaskId#Axo_None;
                _AxisReference^.Telegram111_Out.STW1.activateTraversing := FALSE;
                MC_MoveRelativeErrorID := DINT#0;
                MC_MoveRelativeCycle := ULINT#0;
                State := UINT#0;
                THIS.UpdateOutputs(AxisRef);
            END_IF;

            ErrorID := MC_MoveRelativeErrorID;
            MC_MoveRelativeExecute_PV := Execute;
        END_METHOD

        ///<summary>
        /// This method commands a controlled motion of a specified relative distance additional to the most recent
        /// commanded position in the axis state ‘DiscreteMotion’. The most recent commanded position may be the result of a
        /// previous MC_MoveAdditive motion which was aborted. If the method is activated in the axis state ‘ContinuousMotion’, the
        /// specified relative distance is added to the set position at the time of the execution.
        ///</summary>
        VAR INTERNAL
            MC_MoveAdditiveExecute_PV					: 	BOOL;				//Execute - previous value
            MC_MoveAdditiveErrorID					    : 	DINT;
            MC_MoveAdditiveCycle					    : 	ULINT;
            MC_MoveAdditiveContinuousUpdate_SV          :   BOOL;
            MC_MoveAdditiveDistance_PV                  :   LREAL;
            MC_MoveAdditiveVelocity_PV                  :   LREAL;
            MC_MoveAdditiveAcceleration_PV              :   LREAL;
            MC_MoveAdditiveDeceleration_PV              :   LREAL;
            MC_MoveAdditiveJerk_PV                      :   LREAL;
        END_VAR
        METHOD PUBLIC OVERRIDE MC_MoveAdditive
            VAR_INPUT
                AxisRef         :   AXOpen.Components.Abstractions.Drives.IAxoAxisReference;
                Execute         :   BOOL;                       //  Start the motion at rising edge
                ContinuousUpdate:   BOOL;                       //  Activate ‘ContinuousUpdate’ - target parameters should be changed during movement
                Distance        :   LREAL;                      //  Relative distance for the motion (in technical unit [u]
                Velocity        :   LREAL;                      //  Value of the maximum ‘Velocity’ (not necessarily reached) [u/s].
                Acceleration    :   LREAL;                      //  Value of the ‘Acceleration’ (always positive) (increasing energy of the motor) [u/s2]
                Deceleration    :   LREAL;                      //  Value of the ‘Deceleration’ (always positive) (decreasing energy of the motor) [u/s2]
                Jerk            :   LREAL;                      //  Value of the ‘Jerk’ [u/s3]
            END_VAR
            VAR_OUTPUT
                Done            :   BOOL;                       // Commanded distance reached
                Busy            :   BOOL;                       // The method is not finished and new output values are to be expected
                Active          :   BOOL;                       // Indicates that the method has control on the axis
                CommandAborted  :   BOOL;                       // ‘Command’ is aborted by another command
                Error           :   BOOL;                       // Signals that an error has occurred within the method
                ErrorID         :   DINT;                       // Error identification
            END_VAR
            VAR
                _AxisReference :  REF_TO AXOpen.Components.Festo.Drives.AxoCmmtAsAxisReference;
                Dummy : BOOL;
            END_VAR

            _AxisReference ?= AxisRef;

            IF(_AxisReference = NULL) THEN
                Messenger.Activate(     UINT#1510, eAxoMessageCategory#ProgrammingError);
                DriveStatus.Error.Id := UINT#1510;
                RETURN;
            END_IF;

            Messenger.ActivateOnCondition(ULINT#1511, Execute AND Velocity <= 0, eAxoMessageCategory#ProgrammingError);
            Messenger.ActivateOnCondition(ULINT#1512, Execute AND Acceleration <= 0, eAxoMessageCategory#ProgrammingError);
            Messenger.ActivateOnCondition(ULINT#1513, Execute AND Deceleration <= 0, eAxoMessageCategory#ProgrammingError);
            Messenger.ActivateOnCondition(ULINT#1514, Execute AND Jerk <= 0, eAxoMessageCategory#ProgrammingError);

            IF Execute AND NOT MC_MoveAdditiveExecute_PV THEN
                State := UINT#0;
            END_IF;

            IF Execute THEN
                THIS.UpdateInputs(AxisRef);
                IF NOT ContinuousUpdate THEN
                    MC_MoveAdditiveContinuousUpdate_SV := FALSE;
                END_IF;

                IF State = UINT#0 THEN
                    Busy := TRUE;
                    Active := TRUE;
                    MC_MoveAdditiveErrorID := DINT#0;
                    _AxisReference^.Telegram111_Out.STW1.StartHoming := FALSE;
                    // _AxisReference^.Telegram111_Out.POS_STW1.MDI_MOD := FALSE;
                    _AxisReference^.Telegram111_Out.POS_STW1.PosModulo := FALSE;
                    _AxisReference^.Telegram111_Out.POS_STW1.NegModulo := FALSE;
                    _AxisReference^.Telegram111_Out.POS_STW1.SetupMode := FALSE;
                    // _AxisReference^.Telegram111_Out.POS_STW1.MDI_Activate := FALSE;
                    _AxisReference^.Telegram111_Out.POS_STW2.Trackingmode := FALSE;
                    _AxisReference^.Telegram111_Out.POS_STW2.jog_inc := FALSE;
                    _AxisReference^.Telegram111_Out.POS_STW1.travBlockBit0 := FALSE;
                    _AxisReference^.Telegram111_Out.POS_STW1.travBlockBit1 := FALSE;
                    _AxisReference^.Telegram111_Out.POS_STW1.travBlockBit2 := FALSE;
                    _AxisReference^.Telegram111_Out.POS_STW1.travBlockBit3 := FALSE;
                    _AxisReference^.Telegram111_Out.POS_STW1.travBlockBit4 := FALSE;
                    _AxisReference^.Telegram111_Out.POS_STW1.travBlockBit5 := FALSE;
                    _AxisReference^.Telegram111_Out.POS_STW1.travBlockBit6 := FALSE;
                    _AxisReference^.Telegram111_Out.STW2.TravelToFixStop := FALSE;
                    Parametrization.Inputs.Enable := FALSE;

                    Parametrization.Inputs.Enable := FALSE;
                    MC_MoveAdditiveContinuousUpdate_SV := ContinuousUpdate;
                    IF Velocity > 0 AND Acceleration > 0 AND Deceleration >0 AND Jerk > 0 THEN
                        MC_MoveAdditiveDistance_PV      :=  Distance;
                        MC_MoveAdditiveVelocity_PV      :=  Velocity;
                        MC_MoveAdditiveAcceleration_PV  :=  Acceleration;
                        MC_MoveAdditiveDeceleration_PV  :=  Deceleration;
                        MC_MoveAdditiveJerk_PV          :=  Jerk;
                        _AxisReference^.Telegram111_Out.STW1.activateTraversing := FALSE;
                        IF _AxisReference^.Status.CurrentMotionTaskId = eAxoMotionTaskId#Axo_MoveAbsolute THEN
                            AxoMoveAbsolute_Task.Abort();
                            _AxisReference^.Telegram111_Out.MDI_TARPOS :=   TO_DINT((MC_MoveAbsolutePosition_PV + Distance) * ScalingConstantRequiredPosition);
                            _AxisReference^.Telegram111_Out.MDI_VELOCITY := TO_DINT(Velocity        *   ScalingConstantRequiredVelocity     * _AxisReference^.Data.OverrideVelocityFactor);
                            _AxisReference^.Telegram111_Out.MDI_ACC :=      TO_UINT(Acceleration    *   ScalingConstantRequiredAcceleration * _AxisReference^.Data.OverrideAccelerationFactor);
                            _AxisReference^.Telegram111_Out.MDI_DEC :=      TO_UINT(Deceleration    *   ScalingConstantRequiredDeceleration * _AxisReference^.Data.OverrideAccelerationFactor);
                        ELSE
                            _AxisReference^.Telegram111_Out.MDI_TARPOS :=   TO_DINT((Distance)      *    ScalingConstantRequiredPosition);
                            _AxisReference^.Telegram111_Out.MDI_VELOCITY := TO_DINT(Velocity        *   ScalingConstantRequiredVelocity     * _AxisReference^.Data.OverrideVelocityFactor);
                            _AxisReference^.Telegram111_Out.MDI_ACC :=      TO_UINT(Acceleration    *   ScalingConstantRequiredAcceleration * _AxisReference^.Data.OverrideAccelerationFactor);
                            _AxisReference^.Telegram111_Out.MDI_DEC :=      TO_UINT(Deceleration    *   ScalingConstantRequiredDeceleration * _AxisReference^.Data.OverrideAccelerationFactor);
                            _AxisReference^.Telegram111_Out.POS_STW1.MDI_MOD := FALSE;
                        END_IF;
                        IF _AxisReference^.Status.CurrentMotionTaskId = eAxoMotionTaskId#Axo_MoveRelative THEN
                            AxoMoveRelative_Task.Abort();
                        END_IF;
                        _AxisReference^.Status.CurrentMotionTaskId := eAxoMotionTaskId#Axo_MoveAdditive;
                        _AxisReference^.Data.Cycle := _AxisReference^.Data.Cycle + ULINT#2;
                        MC_MoveAdditiveCycle := _AxisReference^.Data.Cycle ;
                        State := UINT#101;
                    END_IF;
                END_IF;
                IF State = UINT#100 THEN
                    State := UINT#101;
                END_IF;
                //Writing PNU 12327 Jerk
                IF State = UINT#101 THEN
                    Busy := TRUE;
                    Active := TRUE;
                    Parametrization.Inputs.Enable := TRUE;
                    Parametrization.Inputs.ReadWrite   := TRUE;
                    Parametrization.Inputs.ParameterNo := 12327;
                    Parametrization.Inputs.Subindex    := 0;
                    Parametrization.Inputs.AxisNo  := BYTE#1;
                    Parametrization.Inputs.HardwareId  := _AxisReference^.HWIDs.HW_ModuleAccessPoint;
                    Parametrization.Inputs.ValueWriteREAL := TO_REAL(MC_MoveAdditiveJerk_PV  * ScalingConstantRequiredJerk * _AxisReference^.Data.OverrideJerkFactor);
                    IF Parametrization.Outputs.Done AND NOT Parametrization.Outputs.Error THEN
                        State := UINT#102;
                    END_IF;
                    IF Parametrization.Outputs.Error THEN
                        Messenger.Activate(         UINT#1515, eAxoMessageCategory#Error);
                        MC_MoveAdditiveErrorID :=   DINT#1515;
                        State := UINT#109;
                    END_IF;
                END_IF;
                IF State = UINT#102 THEN
                    Busy := TRUE;
                    Active := TRUE;
                    Parametrization.Inputs.Enable := FALSE;
                    Parametrization.Inputs.ReadWrite   := FALSE;
                    IF  NOT Parametrization.Outputs.Done THEN
                        State := UINT#103;
                    END_IF;
                END_IF;
                //Executing movement
                IF State = UINT#103 THEN
                    _AxisReference^.Telegram111_Out.POS_STW1.MDI_Activate := TRUE;
                    _AxisReference^.Telegram111_Out.STW1.activateTraversing := TRUE;
                    IF _AxisReference^.Telegram111_In.ZSW1.acknowledgeTraversingBlockActivated THEN
                        State := UINT#104;
                    END_IF;
                END_IF;
                IF State = UINT#104 THEN
                    _AxisReference^.Telegram111_Out.STW1.activateTraversing := FALSE;
                    IF _AxisReference^.Telegram111_In.ZSW1.targetPosReached THEN
                        State := UINT#105;
                    END_IF;
                END_IF;
                IF State = UINT#105 THEN
                    IF TRUE THEN
                        State := UINT#106;
                    END_IF;
                END_IF;
                IF State = UINT#106 THEN
                    IF TRUE THEN
                        State := UINT#107;
                    END_IF;
                END_IF;
                IF State = UINT#107 THEN
                    Done := TRUE;
                    MC_MoveAdditiveCycle := ULINT#0;
                END_IF;
                IF State = UINT#108 THEN
                    CommandAborted := TRUE;
                END_IF;
                IF State = UINT#109 THEN
                    MC_MoveAdditiveCycle := ULINT#0;
                    Error := TRUE;
                END_IF;

                IF State>=UINT#100 AND State<UINT#107 THEN
                    IF MC_MoveAdditiveContinuousUpdate_SV AND (
                        MC_MoveAdditiveDistance_PV      <>  Distance OR
                        MC_MoveAdditiveVelocity_PV      <>  Velocity OR
                        MC_MoveAdditiveAcceleration_PV  <>  Acceleration OR
                        MC_MoveAdditiveDeceleration_PV  <>  Deceleration OR
                        MC_MoveAdditiveJerk_PV          <>  Jerk ) THEN
                        _AxisReference^.Telegram111_Out.STW1.activateTraversing := FALSE;
                        IF NOT _AxisReference^.Telegram111_In.ZSW1.acknowledgeTraversingBlockActivated THEN
                            IF _AxisReference^.Telegram111_Out.POS_STW1.MDI_MOD THEN
                                _AxisReference^.Telegram111_Out.MDI_TARPOS := _AxisReference^.Telegram111_Out.MDI_TARPOS  + TO_DINT((Distance - MC_MoveAdditiveDistance_PV) * ScalingConstantRequiredPosition);
                            ELSE
                                _AxisReference^.Telegram111_Out.MDI_TARPOS := TO_DINT((Distance) * ScalingConstantRequiredPosition) - _AxisReference^.Telegram111_In.XIST_A;
                            END_IF;
                            _AxisReference^.Telegram111_Out.MDI_VELOCITY := TO_DINT(Velocity        *   ScalingConstantRequiredVelocity     * _AxisReference^.Data.OverrideVelocityFactor);
                            _AxisReference^.Telegram111_Out.MDI_ACC :=      TO_UINT(Acceleration    *   ScalingConstantRequiredAcceleration * _AxisReference^.Data.OverrideAccelerationFactor);
                            _AxisReference^.Telegram111_Out.MDI_DEC :=      TO_UINT(Deceleration    *   ScalingConstantRequiredDeceleration * _AxisReference^.Data.OverrideAccelerationFactor);
                            MC_MoveAdditiveDistance_PV      :=  Distance;
                            MC_MoveAdditiveVelocity_PV      :=  Velocity;
                            MC_MoveAdditiveAcceleration_PV  :=  Acceleration;
                            MC_MoveAdditiveDeceleration_PV  :=  Deceleration;
                            MC_MoveAdditiveJerk_PV          :=  Jerk;
                            State := UINT#101;
                        END_IF;
                    END_IF;
                    IF NOT _AxisReference^.Telegram111_In.ZSW1.operationEnabled THEN
                        State := UINT#108;
                    ELSIF _AxisReference^.Telegram111_In.ZSW1.faultPresent THEN
                        IF MC_MoveAdditiveErrorID = DINT#0 THEN
                            MC_MoveAdditiveErrorID := TO_DINT(_AxisReference^.Telegram111_In.Fault_Code);
                        END_IF;
                        State := UINT#109;
                    ELSIF _AxisReference^.Data.Cycle <> MC_MoveAdditiveCycle THEN
                        _AxisReference^.Data.Cycle := _AxisReference^.Data.Cycle - ULINT#1;
                        State := UINT#108;
                    END_IF;
                END_IF;
                THIS.UpdateOutputs(AxisRef);
            END_IF;

            IF THIS.AxoMoveAdditive_Task.DoneReached() THEN
                _AxisReference^.Status.CurrentMotionTaskId := AXOpen.Components.Drives.eAxoMotionTaskId#Axo_Done;
                _AxisReference^.Telegram111_Out.STW1.activateTraversing := FALSE;
                MC_MoveAdditiveErrorID := DINT#0;
                // MC_MoveAdditiveCycle := ULINT#0;
                State := UINT#0;
                THIS.UpdateOutputs(AxisRef);
            END_IF;

            IF THIS.AxoMoveAdditive_Task.RestoreTriggered() AND State>=UINT#100 AND State<=UINT#109 THEN
                _AxisReference^.Status.CurrentMotionTaskId := AXOpen.Components.Drives.eAxoMotionTaskId#Axo_None;
                _AxisReference^.Telegram111_Out.STW1.activateTraversing := FALSE;
                MC_MoveAdditiveErrorID := DINT#0;
                MC_MoveAdditiveCycle := ULINT#0;
                State := UINT#0;
                THIS.UpdateOutputs(AxisRef);
            END_IF;

            ErrorID := MC_MoveAdditiveErrorID;
            MC_MoveAdditiveExecute_PV := Execute;
        END_METHOD

        ///<summary>
        /// This method commands a never ending controlled motion at a specified velocity.
        ///</summary>
        VAR INTERNAL
            MC_MoveVelocityExecute_PV					: 	BOOL;				//Execute - previous value
            MC_MoveVelocityErrorID					    : 	DINT;
            MC_MoveVelocityCycle					    : 	ULINT;
            MC_MoveVelocityContinuousUpdate_SV          :   BOOL;
            MC_MoveVelocityVelocity_PV                  :   LREAL;
            MC_MoveVelocityAcceleration_PV              :   LREAL;
            MC_MoveVelocityDeceleration_PV              :   LREAL;
            MC_MoveVelocityJerk_PV                      :   LREAL;
            MC_MoveVelocityDirection_PV                 :   AXOpen.Components.Abstractions.Drives.eAxoDriveDirection;
        END_VAR
        METHOD PUBLIC OVERRIDE MC_MoveVelocity
            VAR_INPUT
                AxisRef         :   AXOpen.Components.Abstractions.Drives.IAxoAxisReference;
                Execute         :   BOOL;                       //  Start the motion at rising edge
                ContinuousUpdate:   BOOL;                       //  Activate ‘ContinuousUpdate’ - target parameters should be changed during movement
                Velocity        :   LREAL;                      //  Value of the maximum velocity [u/s]. Can be a signed value.
                Acceleration    :   LREAL;                      //  Value of the ‘Acceleration’ (always positive) (increasing energy of the motor) [u/s2]
                Deceleration    :   LREAL;                      //  Value of the ‘Deceleration’ (always positive) (decreasing energy of the motor) [u/s2]
                Jerk            :   LREAL;                      //  Value of the ‘Jerk’ [u/s3]
                Direction       :   AXOpen.Components.Abstractions.Drives.eAxoDriveDirection;         //  Enum type (1-of-3 values: PositiveDirection, NegativeDirection, and CurrentDirection. Note: shortest way not applicable)
            END_VAR
            VAR_OUTPUT
                InVelocity      :   BOOL;                       // Commanded velocity reached
                Busy            :   BOOL;                       // The method is not finished and new output values are to be expected
                Active          :   BOOL;                       // Indicates that the method has control on the axis
                CommandAborted  :   BOOL;                       // ‘Command’ is aborted by another command
                Error           :   BOOL;                       // Signals that an error has occurred within the method
                ErrorID         :   DINT;                       // Error identification
            END_VAR
            VAR
                _AxisReference :  REF_TO AXOpen.Components.Festo.Drives.AxoCmmtAsAxisReference;
                Dummy : BOOL;
                Velocity_   :   LREAL;
                Direction_  :   AXOpen.Components.Abstractions.Drives.eAxoDriveDirection;
                VelocityWindowPerCent     :   LREAL := LREAL#5.0;
                VelocityWindowMin         :   LREAL;
                VelocityWindowMax         :   LREAL;
            END_VAR

            _AxisReference ?= AxisRef;

            IF(_AxisReference = NULL) THEN
                Messenger.Activate(     UINT#1520, eAxoMessageCategory#ProgrammingError);
                DriveStatus.Error.Id := UINT#1520;
                InVelocity := FALSE;
                RETURN;
            END_IF;

            Messenger.ActivateOnCondition(ULINT#1522, Execute AND Velocity = 0, eAxoMessageCategory#ProgrammingError);
            Messenger.ActivateOnCondition(ULINT#1523, Execute AND Acceleration <= 0, eAxoMessageCategory#ProgrammingError);
            Messenger.ActivateOnCondition(ULINT#1524, Execute AND Deceleration <= 0, eAxoMessageCategory#ProgrammingError);
            Messenger.ActivateOnCondition(ULINT#1525, Execute AND Jerk <= 0, eAxoMessageCategory#ProgrammingError);

            IF THIS.AxoMoveVelocity_Task.StartTriggered()  THEN
                _AxisReference^.Status.CurrentMotionTaskId := AXOpen.Components.Drives.eAxoMotionTaskId#Axo_MoveVelocity;
            END_IF;

            IF Execute AND NOT MC_MoveVelocityExecute_PV AND State = UINT#0 THEN
                _AxisReference^.Data.Cycle := _AxisReference^.Data.Cycle + ULINT#2;
                MC_MoveVelocityCycle := _AxisReference^.Data.Cycle ;
            END_IF;

            IF Execute THEN
                IF Direction <> AXOpen.Components.Abstractions.Drives.eAxoDriveDirection#PositiveDirection AND Direction <> AXOpen.Components.Abstractions.Drives.eAxoDriveDirection#NegativeDirection THEN
                    Messenger.Activate(     UINT#1521, eAxoMessageCategory#ProgrammingError);
                    DriveStatus.Error.Id := UINT#1521;
                    InVelocity := FALSE;
                    RETURN;
                END_IF;

                IF Direction = AXOpen.Components.Abstractions.Drives.eAxoDriveDirection#PositiveDirection THEN
                    Velocity_ := Velocity;
                ELSIF Direction = AXOpen.Components.Abstractions.Drives.eAxoDriveDirection#NegativeDirection THEN
                    Velocity_ := -1 * Velocity;
                ELSE
                    RETURN;
                END_IF;

                IF Velocity_> 0 THEN
                    Direction_ := AXOpen.Components.Abstractions.Drives.eAxoDriveDirection#PositiveDirection;
                ELSE
                    Direction_ := AXOpen.Components.Abstractions.Drives.eAxoDriveDirection#NegativeDirection;
                END_IF;

                THIS.UpdateInputs(AxisRef);
                IF NOT ContinuousUpdate THEN
                    MC_MoveVelocityContinuousUpdate_SV := FALSE;
                END_IF;

                IF State = UINT#0 THEN
                    Busy := TRUE;
                    Active := TRUE;
                    MC_MoveVelocityErrorID := DINT#0;
                    _AxisReference^.Telegram111_Out.STW1.StartHoming := FALSE;
                    _AxisReference^.Telegram111_Out.POS_STW1.MDI_MOD := FALSE;
                    _AxisReference^.Telegram111_Out.POS_STW1.PosModulo := FALSE;
                    _AxisReference^.Telegram111_Out.POS_STW1.NegModulo := FALSE;
                    _AxisReference^.Telegram111_Out.POS_STW1.SetupMode := FALSE;
                    _AxisReference^.Telegram111_Out.POS_STW1.MDI_Activate := FALSE;
                    _AxisReference^.Telegram111_Out.POS_STW2.Trackingmode := FALSE;
                    _AxisReference^.Telegram111_Out.POS_STW2.jog_inc := FALSE;
                    _AxisReference^.Telegram111_Out.POS_STW1.travBlockBit0 := FALSE;
                    _AxisReference^.Telegram111_Out.POS_STW1.travBlockBit1 := FALSE;
                    _AxisReference^.Telegram111_Out.POS_STW1.travBlockBit2 := FALSE;
                    _AxisReference^.Telegram111_Out.POS_STW1.travBlockBit3 := FALSE;
                    _AxisReference^.Telegram111_Out.POS_STW1.travBlockBit4 := FALSE;
                    _AxisReference^.Telegram111_Out.POS_STW1.travBlockBit5 := FALSE;
                    _AxisReference^.Telegram111_Out.POS_STW1.travBlockBit6 := FALSE;
                    _AxisReference^.Telegram111_Out.STW2.TravelToFixStop := FALSE;
                    Parametrization.Inputs.Enable := FALSE;
                    MC_MoveVelocityContinuousUpdate_SV := ContinuousUpdate;
                    State := UINT#110;
                END_IF;
                IF State = UINT#110 THEN
                    Busy := TRUE;
                    Active := TRUE;
                    IF Velocity <> 0 AND Acceleration > 0 AND Deceleration >0 AND Jerk > 0 THEN
                        _AxisReference^.Telegram111_Out.MDI_TARPOS := DINT#0;
                        _AxisReference^.Telegram111_Out.MDI_VELOCITY := TO_DINT(ABS(Velocity_)  *   ScalingConstantRequiredVelocity     * _AxisReference^.Data.OverrideVelocityFactor);
                        _AxisReference^.Telegram111_Out.MDI_ACC :=      TO_UINT(Acceleration    *   ScalingConstantRequiredAcceleration * _AxisReference^.Data.OverrideAccelerationFactor);
                        _AxisReference^.Telegram111_Out.MDI_DEC :=      TO_UINT(Deceleration    *   ScalingConstantRequiredDeceleration * _AxisReference^.Data.OverrideAccelerationFactor);

                        MC_MoveVelocityVelocity_PV      :=  Velocity_;
                        MC_MoveVelocityAcceleration_PV  :=  Acceleration;
                        MC_MoveVelocityDeceleration_PV  :=  Deceleration;
                        MC_MoveVelocityJerk_PV          :=  Jerk;
                        MC_MoveVelocityDirection_PV     :=  Direction_;
                        State := UINT#111;
                    END_IF;
                END_IF;
                //Writing PNU 12327 Jerk
                IF State = UINT#111 THEN
                    Busy := TRUE;
                    Active := TRUE;
                    Parametrization.Inputs.Enable := TRUE;
                    Parametrization.Inputs.ReadWrite   := TRUE;
                    Parametrization.Inputs.ParameterNo := 12327;
                    Parametrization.Inputs.Subindex    := 0;
                    Parametrization.Inputs.AxisNo  := BYTE#1;
                    Parametrization.Inputs.HardwareId  := _AxisReference^.HWIDs.HW_ModuleAccessPoint;
                    Parametrization.Inputs.ValueWriteREAL := TO_REAL(MC_MoveVelocityJerk_PV * ScalingConstantRequiredJerk * _AxisReference^.Data.OverrideJerkFactor);
                    IF Parametrization.Outputs.Done AND NOT Parametrization.Outputs.Error THEN
                        State := UINT#112;
                    END_IF;
                    IF Parametrization.Outputs.Error THEN
                        Messenger.Activate(         UINT#1526, eAxoMessageCategory#Error);
                        MC_MoveVelocityErrorID :=   DINT#1526;
                        State := UINT#119;
                    END_IF;
                END_IF;
                IF State = UINT#112 THEN
                    Busy := TRUE;
                    Active := TRUE;
                    Parametrization.Inputs.Enable := FALSE;
                    Parametrization.Inputs.ReadWrite   := FALSE;
                    IF  NOT Parametrization.Outputs.Done THEN
                        State := UINT#113;
                    END_IF;
                END_IF;
                //Executing movement
                IF State = UINT#113 THEN
                    _AxisReference^.Telegram111_Out.POS_STW1.MDI_Activate := TRUE;
                    _AxisReference^.Telegram111_Out.POS_STW1.MDI_MOD := TRUE;
                    _AxisReference^.Telegram111_Out.POS_STW1.SetupMode := TRUE;
                    _AxisReference^.Telegram111_Out.POS_STW1.PosModulo := Direction_ = AXOpen.Components.Abstractions.Drives.eAxoDriveDirection#PositiveDirection;
                    _AxisReference^.Telegram111_Out.POS_STW1.NegModulo := Direction_ = AXOpen.Components.Abstractions.Drives.eAxoDriveDirection#NegativeDirection;
                    _AxisReference^.Telegram111_Out.STW1.activateTraversing := TRUE;

                    IF _AxisReference^.Telegram111_In.ZSW1.acknowledgeTraversingBlockActivated THEN
                        State := UINT#114;
                    END_IF;
                END_IF;
                IF State = UINT#114 THEN
                    // _AxisReference^.Telegram111_Out.STW1.activateTraversing := FALSE;
                    IF NOT _AxisReference^.Telegram111_In.ZSW1.targetPosReached  AND NOT _AxisReference^.Telegram111_In.ZSW1.axisAccelerates THEN
                        State := UINT#115;
                    END_IF;
                END_IF;
                IF Direction_ = AXOpen.Components.Abstractions.Drives.eAxoDriveDirection#PositiveDirection  THEN
                    VelocityWindowMax := Velocity_ + (Velocity_ * VelocityWindowPerCent / REAL#100.0);
                    VelocityWindowMin := Velocity_ - (Velocity_ * VelocityWindowPerCent / REAL#100.0);
                ELSE
                    VelocityWindowMax := Velocity_ - (Velocity_ * VelocityWindowPerCent / REAL#100.0);
                    VelocityWindowMin := Velocity_ + (Velocity_ * VelocityWindowPerCent / REAL#100.0);
                END_IF;
                InVelocity := ActualVelocity >= VelocityWindowMin AND ActualVelocity <= VelocityWindowMax;
                IF State = UINT#115 THEN
                    IF InVelocity THEN
                        State := UINT#116;
                    END_IF;
                END_IF;
                IF State = UINT#116 THEN
                    IF NOT MC_MoveVelocityContinuousUpdate_SV THEN
                        State := UINT#117;
                    END_IF;
                END_IF;
                IF State = UINT#117 THEN
                    InVelocity := TRUE;
                    MC_MoveVelocityCycle := ULINT#0;
                END_IF;
                IF State = UINT#118 THEN
                    CommandAborted := TRUE;
                END_IF;
                IF State = UINT#119 THEN
                    MC_MoveVelocityCycle := ULINT#0;
                    Error := TRUE;
                END_IF;

                IF State>=UINT#110 AND State<UINT#117 THEN
                    IF MC_MoveVelocityContinuousUpdate_SV AND (
                        MC_MoveVelocityVelocity_PV      <>  Velocity_ OR
                        MC_MoveVelocityAcceleration_PV  <>  Acceleration OR
                        MC_MoveVelocityDeceleration_PV  <>  Deceleration OR
                        MC_MoveVelocityJerk_PV          <>  Jerk OR
                        MC_MoveVelocityDirection_PV     <>  Direction_ ) THEN
                        _AxisReference^.Telegram111_Out.STW1.activateTraversing := FALSE;
                        IF NOT _AxisReference^.Telegram111_In.ZSW1.acknowledgeTraversingBlockActivated THEN
                            State := UINT#110;
                        END_IF;
                    END_IF;
                    IF NOT _AxisReference^.Telegram111_In.ZSW1.operationEnabled THEN
                        State := UINT#118;
                    ELSIF _AxisReference^.Telegram111_In.ZSW1.faultPresent THEN
                        IF MC_MoveVelocityErrorID = DINT#0 THEN
                            MC_MoveVelocityErrorID := TO_DINT(_AxisReference^.Telegram111_In.Fault_Code);
                        END_IF;
                        State := UINT#119;
                    ELSIF _AxisReference^.Data.Cycle <> MC_MoveVelocityCycle THEN
                        _AxisReference^.Data.Cycle := _AxisReference^.Data.Cycle - ULINT#1;
                        State := UINT#118;
                    END_IF;
                END_IF;
                THIS.UpdateOutputs(AxisRef);
            END_IF;

            IF THIS.AxoMoveVelocity_Task.DoneReached() THEN
                _AxisReference^.Status.CurrentMotionTaskId := AXOpen.Components.Drives.eAxoMotionTaskId#Axo_Done;
                _AxisReference^.Telegram111_Out.STW1.activateTraversing := FALSE;
                MC_MoveVelocityErrorID := DINT#0;
                // MC_MoveVelocityCycle := ULINT#0;
                State := UINT#0;
                THIS.UpdateOutputs(AxisRef);
            END_IF;

            IF THIS.AxoMoveVelocity_Task.RestoreTriggered() AND State>=UINT#110 AND State<=UINT#119 THEN
                _AxisReference^.Status.CurrentMotionTaskId := AXOpen.Components.Drives.eAxoMotionTaskId#Axo_None;
                _AxisReference^.Telegram111_Out.STW1.activateTraversing := FALSE;
                MC_MoveVelocityErrorID := DINT#0;
                MC_MoveVelocityCycle := ULINT#0;
                State := UINT#0;
                THIS.UpdateOutputs(AxisRef);
            END_IF;

            ErrorID := MC_MoveVelocityErrorID;
            MC_MoveVelocityExecute_PV := Execute;
        END_METHOD

        ///<summary>
        /// This method continuously exerts a torque or force of the specified magnitude. This magnitude is
        /// approached using a defined ramp (‘TorqueRamp’), and the method sets the ‘InTorque’ output if the
        /// commanded torque level is reached. This method is applicable for force and torque. When there is no external
        /// load, force is applicable. Positive torque is in the positive direction of velocity.
        ///</summary>
        VAR INTERNAL
            MC_TorqueControlExecute_PV					: 	BOOL;				//Execute - previous value
            MC_TorqueControlErrorID					    : 	DINT;
            MC_TorqueControlCycle					    : 	ULINT;
            MC_TorqueControlContinuousUpdate_SV         :   BOOL;
            MC_TorqueControlTorque_PV                   :   LREAL;
            MC_TorqueControlTorqueRamp_PV               :   LREAL;
            MC_TorqueControlPositionLimit_PV            :   LREAL;
            MC_TorqueControlVelocity_PV                 :   LREAL;
            MC_TorqueControlAcceleration_PV             :   LREAL;
            MC_TorqueControlDeceleration_PV             :   LREAL;
            MC_TorqueControlJerk_PV                     :   LREAL;
            MC_TorqueControlDirection_PV                :   AXOpen.Components.Abstractions.Drives.eAxoDriveDirection;
            MC_TorqueControlTorqueA                     :   LREAL;
            MC_TorqueControlPositiveDirectionA          :   BOOL;
            MC_TorqueControlTorqueWindowMin             :   LREAL;
            MC_TorqueControlTorqueWindowMax             :   LREAL;
            MC_TorqueControlTorqueWindowTimer           :   AXOpen.Timers.OnDelayTimer;

        END_VAR
        METHOD PUBLIC OVERRIDE MC_TorqueControl
            VAR_INPUT
                AxisRef         :   AXOpen.Components.Abstractions.Drives.IAxoAxisReference;
                Execute         :   BOOL;                       //  Start the motion at rising edge
                ContinuousUpdate:   BOOL;                       //  Activate ‘ContinuousUpdate’ - target parameters should be changed during movement
                Torque          :   LREAL;                      //  Value of the torque (Torque or force in technical unit [u])
                TorqueRamp      :   LREAL;                      //  The maximum time derivative of the set value of the torque or force (in technical unit per sec. [u/s])
                PositionLimit   :   LREAL;                      //  Position limit
                Velocity        :   LREAL;                      //  Absolute value of the maximum velocity.
                Acceleration    :   LREAL;                      //  Value of the maximum acceleration (acceleration is applicable with same sign of torque and velocity)
                Deceleration    :   LREAL;                      //  Value of the maximum deceleration (deceleration is applicable with opposite signs of torque and velocity)
                Jerk            :   LREAL;                      //  Value of the maximum jerk
                Direction       :   AXOpen.Components.Abstractions.Drives.eAxoDriveDirection;         //  Enum type (1 of 2 values: PositiveDirection, NegativeDirection or CurrentDirection). Specifies the direction of the torque. (Note: Torque input can be signed value).
            END_VAR
            VAR_OUTPUT
                InTorque        :   BOOL;                       //  Setpoint value of torque or force equals the commandedvalue
                Busy            :   BOOL;                       //  The method is not finished and new output values are to be expected
                Active          :   BOOL;                       //  Indicates that the method has control on the axis
                CommandAborted  :   BOOL;                       //  ‘Command’ is aborted by another command
                Error           :   BOOL;                       //  Signals that an error has occurred within the method
                ErrorID         :   DINT;                       //  Error identification
            END_VAR
            VAR
                _AxisReference :  REF_TO AXOpen.Components.Festo.Drives.AxoCmmtAsAxisReference;
                Dummy : BOOL;
            END_VAR

            _AxisReference ?= AxisRef;

            IF(_AxisReference = NULL) THEN
                Messenger.Activate(     UINT#1530, eAxoMessageCategory#ProgrammingError);
                DriveStatus.Error.Id := UINT#1530;
                RETURN;
            END_IF;

            IF THIS.AxoTorqueControl_Task.StartTriggered()  THEN
                _AxisReference^.Status.CurrentMotionTaskId := AXOpen.Components.Drives.eAxoMotionTaskId#Axo_TorqueControl;
            END_IF;

            IF Execute AND NOT MC_TorqueControlExecute_PV AND State = UINT#0 THEN
                _AxisReference^.Data.Cycle := _AxisReference^.Data.Cycle + ULINT#2;
                MC_TorqueControlCycle := _AxisReference^.Data.Cycle ;
            END_IF;

            IF Execute THEN
                THIS.UpdateInputs(AxisRef);
                IF NOT ContinuousUpdate THEN
                    MC_TorqueControlContinuousUpdate_SV := FALSE;
                END_IF;

                IF State = UINT#0 THEN
                    Messenger.ActivateOnCondition(ULINT#1531, Direction <> AXOpen.Components.Abstractions.Drives.eAxoDriveDirection#PositiveDirection AND Direction <> AXOpen.Components.Abstractions.Drives.eAxoDriveDirection#NegativeDirection, eAxoMessageCategory#ProgrammingError);
                    Messenger.ActivateOnCondition(ULINT#1532, Execute AND Velocity <= 0, eAxoMessageCategory#ProgrammingError);
                    Messenger.ActivateOnCondition(ULINT#1533, Execute AND Acceleration <= 0, eAxoMessageCategory#ProgrammingError);
                    Messenger.ActivateOnCondition(ULINT#1534, Execute AND Deceleration <= 0, eAxoMessageCategory#ProgrammingError);
                    Messenger.ActivateOnCondition(ULINT#1535, Execute AND Jerk <= 0, eAxoMessageCategory#ProgrammingError);
                    Messenger.ActivateOnCondition(ULINT#1536, Execute AND Torque = 0, eAxoMessageCategory#ProgrammingError);
                    Messenger.ActivateOnCondition(ULINT#1537, Execute AND TorqueRamp <= 0, eAxoMessageCategory#ProgrammingError);

                    IF Direction = AXOpen.Components.Abstractions.Drives.eAxoDriveDirection#PositiveDirection THEN
                        MC_TorqueControlTorqueA := Torque;
                    ELSIF Direction = AXOpen.Components.Abstractions.Drives.eAxoDriveDirection#NegativeDirection THEN
                        MC_TorqueControlTorqueA := -1 * Torque;
                    ELSE
                        RETURN;
                    END_IF;

                    MC_TorqueControlPositiveDirectionA := MC_TorqueControlTorqueA > 0;

                    IF MC_TorqueControlPositiveDirectionA  THEN
                        MC_TorqueControlTorqueWindowMax := MC_TorqueControlTorqueA + (MC_TorqueControlTorqueA * _AxisReference^.Config.InTorqueWindowPerCent / REAL#100.0);
                        MC_TorqueControlTorqueWindowMin := MC_TorqueControlTorqueA - (MC_TorqueControlTorqueA * _AxisReference^.Config.InTorqueWindowPerCent / REAL#100.0);
                    ELSE
                        MC_TorqueControlTorqueWindowMax := MC_TorqueControlTorqueA - (MC_TorqueControlTorqueA * _AxisReference^.Config.InTorqueWindowPerCent / REAL#100.0);
                        MC_TorqueControlTorqueWindowMin := MC_TorqueControlTorqueA + (MC_TorqueControlTorqueA * _AxisReference^.Config.InTorqueWindowPerCent / REAL#100.0);
                    END_IF;

                    Busy := TRUE;
                    Active := TRUE;
                    MC_TorqueControlErrorID := DINT#0;
                    _AxisReference^.Telegram111_Out.STW1.StartHoming := FALSE;
                    _AxisReference^.Telegram111_Out.POS_STW1.MDI_MOD := FALSE;
                    _AxisReference^.Telegram111_Out.POS_STW1.PosModulo := FALSE;
                    _AxisReference^.Telegram111_Out.POS_STW1.NegModulo := FALSE;
                    _AxisReference^.Telegram111_Out.POS_STW1.SetupMode := FALSE;
                    _AxisReference^.Telegram111_Out.POS_STW1.MDI_Activate := FALSE;
                    _AxisReference^.Telegram111_Out.POS_STW2.Trackingmode := FALSE;
                    _AxisReference^.Telegram111_Out.POS_STW2.jog_inc := FALSE;
                    _AxisReference^.Telegram111_Out.POS_STW1.travBlockBit0 := FALSE;
                    _AxisReference^.Telegram111_Out.POS_STW1.travBlockBit1 := FALSE;
                    _AxisReference^.Telegram111_Out.POS_STW1.travBlockBit2 := FALSE;
                    _AxisReference^.Telegram111_Out.POS_STW1.travBlockBit3 := FALSE;
                    _AxisReference^.Telegram111_Out.POS_STW1.travBlockBit4 := FALSE;
                    _AxisReference^.Telegram111_Out.POS_STW1.travBlockBit5 := FALSE;
                    _AxisReference^.Telegram111_Out.POS_STW1.travBlockBit6 := FALSE;
                    _AxisReference^.Telegram111_Out.STW2.TravelToFixStop := FALSE;
                    Parametrization.Inputs.Enable := FALSE;
                    MC_TorqueControlContinuousUpdate_SV := ContinuousUpdate;
                    IF Velocity > 0 AND Acceleration > 0 AND Deceleration > 0 AND Jerk > 0 AND Torque <> 0 AND TorqueRamp > 0 THEN
                        _AxisReference^.Telegram111_Out.MDI_TARPOS :=   TO_DINT(PositionLimit   *   ScalingConstantRequiredPosition);
                        _AxisReference^.Telegram111_Out.MDI_VELOCITY := TO_DINT(Velocity        *   ScalingConstantRequiredVelocity     * _AxisReference^.Data.OverrideVelocityFactor);
                        _AxisReference^.Telegram111_Out.MDI_ACC :=      TO_UINT(Acceleration    *   ScalingConstantRequiredAcceleration * _AxisReference^.Data.OverrideAccelerationFactor);
                        _AxisReference^.Telegram111_Out.MDI_DEC :=      TO_UINT(Deceleration    *   ScalingConstantRequiredDeceleration * _AxisReference^.Data.OverrideAccelerationFactor);
